ABB RobotStudio station: Lab_1_Template.rspag

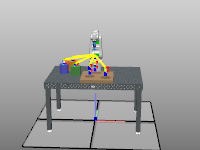
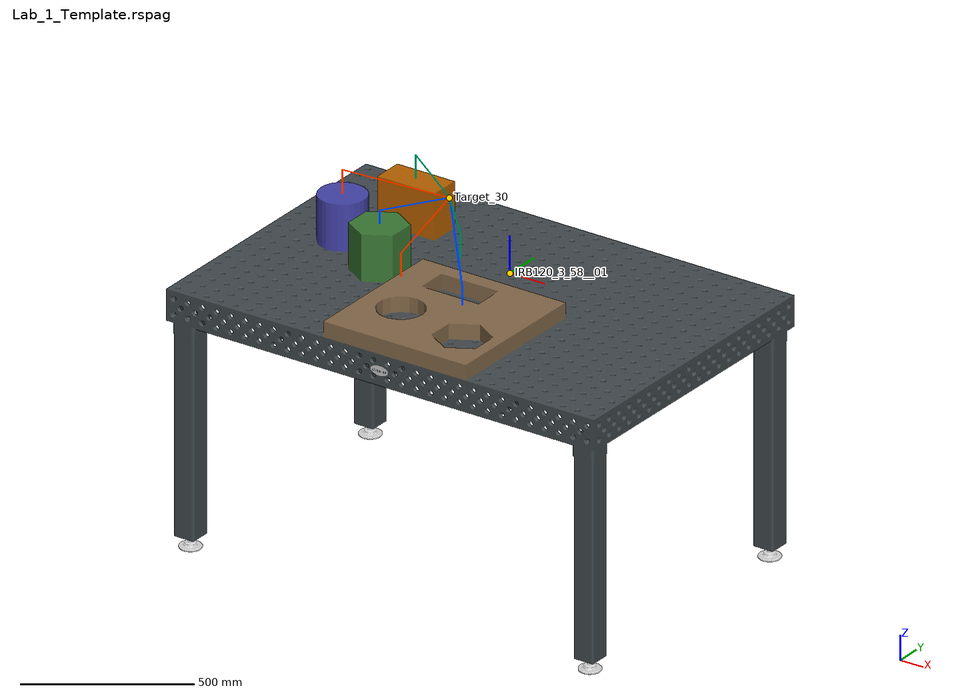
[picture v1: parts stored in the station drawn from their meshes, with robot base, taught points and paths (robot models come from the ABB library and are not in the file)]
--- station ---
Station Solution_1_Tutorial (saved by RobotStudio 21.4.9700.0)
Controller Controller1, task T_ROB1: task frame (RAPID world) sits at (0, 150, 830) mm, rotated rx 0 ry 0 rz -90 deg in the station
Controller Controller1
  mechanical unit ROB_1: IRB120_3_58__01, 6 joints, base frame (0, 0, 0) mm
Layout (positions relative to the parent item):
  - table [part] at (-200, -500, 830) mm, size 500 x 500 x 50 mm
  - object_1 [part] at (-600, -150, 830) mm, size 200 x 100 x 150 mm
  - object_2 [part] at (-650, -150, 830) mm, size 149.5 x 149.7 x 150 mm
  - object_3 [part] at (-700, -200, 830) mm, size 155.5 x 179.5 x 150 mm
  - siegmund_1500_1000 [part], size 1500 x 1010.3 x 830 mm
  - object_11 [part] at (-200, -500, 830) mm, size 200 x 100 x 150 mm
  - object_22 [part] at (-200, -500, 830) mm, size 149.5 x 149.7 x 150 mm
  - object_33 [part] at (-200, -500, 829.48) mm, size 155.5 x 179.5 x 150 mm
  - smc_gripper [mechanism, from Downloads\smc_gripper.rslib] at (0, -152, 1388) mm, rotated rx 180 ry 0 rz 90 deg
  - IRB120_3_58__01 [mechanism, from Robots\IRB120_3_58_G_01.rslib] at (0, 150, 830) mm, rotated rx 0 ry 0 rz -90 deg; joint values [0, 0, 0, 0, 1.5708, 0] (rad or m)
  - Positioner [smart component, from Components\Positioner.rslib] at (0, 0, 0) mm
      properties: Object=object_3; Position=[-0.7 -0.2 0.83]; Orientation=[0 0 0]; Reference=Global; ReferenceObject=(none)
  - Attacher [smart component, from Components\Attacher.rslib]
      properties: Parent=smc_gripper; Flange=0; Child=object_3; Mount=false; Offset=[0 0 0]; Orientation=[0 0 0]
  - Detacher [smart component, from Components\Detacher.rslib]
      properties: Child=object_3; KeepPosition=true
  - Positioner_2 [smart component, from Components\Positioner.rslib]
      properties: Object=object_2; Position=[-0.65 -0.15 0.83]; Orientation=[0 0 0]; Reference=Global; ReferenceObject=(none)
  - Attacher_2 [smart component, from Components\Attacher.rslib]
      properties: Parent=smc_gripper; Flange=0; Child=object_2; Mount=false; Offset=[0 0 0]; Orientation=[0 0 0]
  - Detacher_2 [smart component, from Components\Detacher.rslib]
      properties: Child=object_2; KeepPosition=true
  - Positioner_3 [smart component, from Components\Positioner.rslib]
      properties: Object=object_1; Position=[-0.6 -0.15 0.83]; Orientation=[0 0 0]; Reference=Global; ReferenceObject=(none)
  - Attacher_3 [smart component, from Components\Attacher.rslib]
      properties: Parent=smc_gripper; Flange=0; Child=object_1; Mount=false; Offset=[0 0 0]; Orientation=[0 0 0]
  - Detacher_3 [smart component, from Components\Detacher.rslib]
      properties: Child=object_1; KeepPosition=true
Attachment: smc_gripper is attached to IRB120_3_58__01 / Link6
Attachment: Positioner is attached to object_1
Station signals: DI DI_POS_OBJ_1, DI DI_POS_OBJ_2, DI DI_POS_OBJ_3
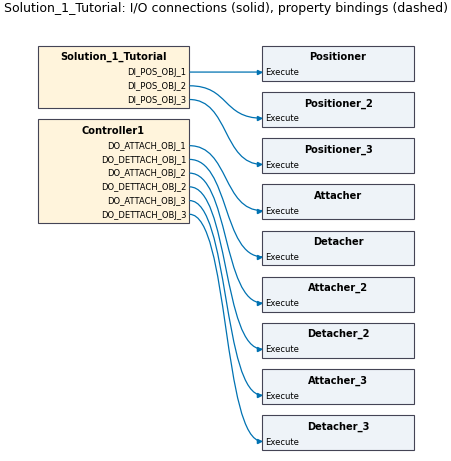
Station logic (signal -> signal, property => property):
  Solution_1_Tutorial.DI_POS_OBJ_1 -> Positioner.Execute
  Controller1.DO_ATTACH_OBJ_1 -> Attacher.Execute
  Controller1.DO_DETTACH_OBJ_1 -> Detacher.Execute
  Solution_1_Tutorial.DI_POS_OBJ_2 -> Positioner_2.Execute
  Controller1.DO_ATTACH_OBJ_2 -> Attacher_2.Execute
  Controller1.DO_DETTACH_OBJ_2 -> Detacher_2.Execute
  Solution_1_Tutorial.DI_POS_OBJ_3 -> Positioner_3.Execute
  Controller1.DO_ATTACH_OBJ_3 -> Attacher_3.Execute
  Controller1.DO_DETTACH_OBJ_3 -> Detacher_3.Execute

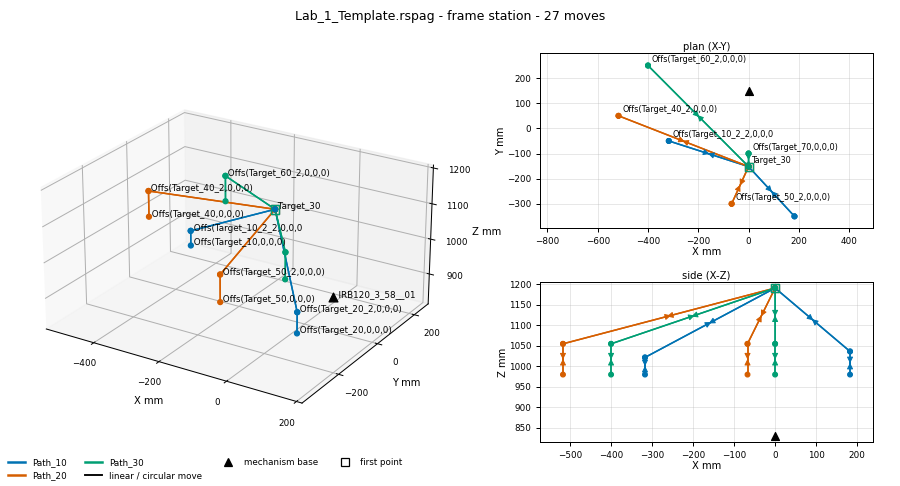
[picture p0: tool path of Lab_1_Template.rspag in frame station, 27 of 27 moves have a stored position in this frame; points joined in program order, loops and branches not executed]
--- Backups/Controller1/RAPID/TASK1/PROGMOD/CalibData.mod ---
MODULE CalibData
    PERS tooldata smc_gripper:=[TRUE,[[0,0.004,197.001],[1,0,0,0]],[1,[0.207,-0.496,71.18],[1,0,0,0],0,0,0]];
ENDMODULE

--- Backups/Controller1/RAPID/TASK1/PROGMOD/Module1.mod ---
MODULE Module1
    CONST robtarget Target_30:=[[302,0.004,360.999],[0,0,1,0],[-1,0,-1,0],[9E+09,9E+09,9E+09,9E+09,9E+09,9E+09]];
    CONST robtarget Target_50_2:=[[450,-67.298,225],[0,0.707106781,0.707106781,0],[-1,0,0,0],[9E+09,9E+09,9E+09,9E+09,9E+09,9E+09]];
    CONST robtarget Target_40_2:=[[100,-517.298,225],[0,0.707106781,0.707106781,0],[-1,0,0,0],[9E+09,9E+09,9E+09,9E+09,9E+09,9E+09]];
    CONST robtarget Target_50:=[[450,-67.298,150],[0,0.707106781,0.707106781,0],[-1,0,0,0],[9E+09,9E+09,9E+09,9E+09,9E+09,9E+09]];
    CONST robtarget Target_40:=[[100,-517.298,150],[0,0.707106781,0.707106781,0],[-1,0,0,0],[9E+09,9E+09,9E+09,9E+09,9E+09,9E+09]];
    CONST robtarget Target_10_2_2:=[[200,-317.298,191.790699476],[0,0.707106781,0.707106781,0],[-1,0,0,0],[9E+09,9E+09,9E+09,9E+09,9E+09,9E+09]];
    CONST robtarget Target_10:=[[200,-317.298,150],[0,0.707106781,0.707106781,0],[0,0,0,0],[9E+09,9E+09,9E+09,9E+09,9E+09,9E+09]];
    CONST robtarget Target_20_2:=[[500,182.702,206.448562902],[0,0.707106781,0.707106781,0],[0,0,0,0],[9E+09,9E+09,9E+09,9E+09,9E+09,9E+09]];
    CONST robtarget Target_20:=[[500,182.702,150],[0,0.707106781,0.707106781,0],[0,0,1,0],[9E+09,9E+09,9E+09,9E+09,9E+09,9E+09]];
    CONST robtarget Target_60_2:=[[-100,-400,225],[0,0.707106781,0.707106781,0],[-2,0,-1,0],[9E+09,9E+09,9E+09,9E+09,9E+09,9E+09]];
    CONST robtarget Target_60:=[[-100,-400,150],[0,0.707106781,0.707106781,0],[-2,0,-1,0],[9E+09,9E+09,9E+09,9E+09,9E+09,9E+09]];
    CONST robtarget Target_70_2:=[[250,0,225],[0,0.707106781,0.707106781,0],[0,0,0,0],[9E+09,9E+09,9E+09,9E+09,9E+09,9E+09]];
    CONST robtarget Target_70:=[[250,0,150],[0,0.707106781,0.707106781,0],[0,0,0,0],[9E+09,9E+09,9E+09,9E+09,9E+09,9E+09]];
!***********************************************************
    !
    ! Module:  Module1
    !
    ! Description:
    !   <Insert description here>
    !
    ! Author: vojta
    !
    ! Version: 1.0
    !
    !***********************************************************


    !***********************************************************
    !
    ! Procedure main
    !
    !   This is the entry point of your program
    !
    !***********************************************************
    PROC main()
       Path_10;
       Path_20;
       Path_30;
    ENDPROC

    PROC Path_10()
        MoveL Target_30,v1000,z100,smc_gripper\WObj:=wobj0;
        !PICK
        MoveL Offs(Target_10_2_2, 0, 0, 0),v200,fine,smc_gripper\WObj:=wobj0;
        MoveL Offs(Target_10, 0, 0, 0),v200,fine,smc_gripper\WObj:=wobj0;
        WaitTime 0.1;
        PulseDO DO_ATTACH_OBJ_1;
        WaitTime 0.1;
        MoveL Offs(Target_10_2_2, 0, 0, 0),v200,fine,smc_gripper\WObj:=wobj0;

        MoveL Target_30,v1000,z100,smc_gripper\WObj:=wobj0;
        !PLACE
        MoveL Offs(Target_20_2, 0, 0, 0),v200,fine,smc_gripper\WObj:=wobj0;
        MoveL Offs(Target_20, 0, 0, 0),v200,fine,smc_gripper\WObj:=wobj0;
        WaitTime 0.1;
        PulseDO DO_DETTACH_OBJ_1;
        WaitTime 0.1;
        MoveL Offs(Target_20_2, 0, 0, 0),v200,fine,smc_gripper\WObj:=wobj0;

        MoveL Target_30,v1000,z100,smc_gripper\WObj:=wobj0;
    ENDPROC

     PROC Path_20()
        MoveL Target_30,v1000,z100,smc_gripper\WObj:=wobj0;
        !PICK
        MoveL Offs(Target_40_2, 0, 0, 0),v200,fine,smc_gripper\WObj:=wobj0;
        MoveL Offs(Target_40, 0, 0, 0),v200,fine,smc_gripper\WObj:=wobj0;
        WaitTime 0.1;
        PulseDO DO_ATTACH_OBJ_2;
        WaitTime 0.1;
        MoveL Offs(Target_40_2, 0, 0, 0),v200,fine,smc_gripper\WObj:=wobj0;

        MoveL Target_30,v1000,z100,smc_gripper\WObj:=wobj0;
        !PLACE
        MoveL Offs(Target_50_2, 0, 0, 0),v200,fine,smc_gripper\WObj:=wobj0;
        MoveL Offs(Target_50, 0, 0, 0),v200,fine,smc_gripper\WObj:=wobj0;
        WaitTime 0.1;
        PulseDO DO_DETTACH_OBJ_2;
        WaitTime 0.1;
        MoveL Offs(Target_50_2, 0, 0, 0),v200,fine,smc_gripper\WObj:=wobj0;

        MoveL Target_30,v1000,z100,smc_gripper\WObj:=wobj0;
    ENDPROC
    PROC Path_30()
        MoveL Target_30,v1000,z100,smc_gripper\WObj:=wobj0;
        !PICK
        MoveL Offs(Target_60_2, 0, 0, 0),v200,fine,smc_gripper\WObj:=wobj0;
        MoveL Offs(Target_60, 0, 0, 0),v200,fine,smc_gripper\WObj:=wobj0;
        WaitTime 0.1;
        PulseDO DO_ATTACH_OBJ_3;
        WaitTime 0.1;
        MoveL Offs(Target_60_2, 0, 0, 0),v200,fine,smc_gripper\WObj:=wobj0;

        MoveL Target_30,v1000,z100,smc_gripper\WObj:=wobj0;
        !PLACE
        MoveL Offs(Target_70_2, 0, 0, 0),v200,fine,smc_gripper\WObj:=wobj0;
        MoveL Offs(Target_70, 0, 0, 0),v200,fine,smc_gripper\WObj:=wobj0;
        WaitTime 0.1;
        PulseDO DO_DETTACH_OBJ_3;
        WaitTime 0.1;
        MoveL Offs(Target_70_2, 0, 0, 0),v200,fine,smc_gripper\WObj:=wobj0;

        MoveL Target_30,v1000,z100,smc_gripper\WObj:=wobj0;
    ENDPROC
ENDMODULE

--- Backups/Controller1/SYSPAR/EIO.cfg ---
EIO:CFG_1.0:6:1::
#
EIO_SIGNAL:

      -Name "DO_ATTACH_OBJ_1" -SignalType "DO"

      -Name "DO_DETTACH_OBJ_1" -SignalType "DO"

      -Name "DO_ATTACH_OBJ_2" -SignalType "DO"

      -Name "DO_DETTACH_OBJ_2" -SignalType "DO"

      -Name "DO_ATTACH_OBJ_3" -SignalType "DO"

      -Name "DO_DETTACH_OBJ_3" -SignalType "DO"
